FUNCTION F_TargetReachedOrHigher : BOOL
VAR_INPUT
	fCurrentPos: LREAL;
	fTargetPos: LREAL;
END_VAR


F_TargetReachedOrHigher := fCurrentPos >= (fTargetPos - fEpsilon);

END_FUNCTION

(* stored: Version 1.1.0.1, ProductVersion 3.1.4022.9
   POU F_TargetReachedOrHigher: Id {714a5ff3-321b-4b6c-8dd8-7ffb4626df7c}, SpecialFunc None *)
